{attribute 'qualified_only'}
{attribute 'strict'}
{attribute 'to_string'}
TYPE E_CabinAirState :
(
	NONE := 0, //Do Nothing
	
	AMBIENT,
	
	FLUSHED
	
	
);
END_TYPE

(* stored: Version 1.1.0.1, ProductVersion 3.1.4024.12
   DUT E_CabinAirState: Id {0ddc39e3-34e6-450a-96d2-841f79219c0f} *)
